GLOBALCONSTANTS DefaultPool (* Global constants *)
  PACKAGE FBs::Counter::const;
  VAR_GLOBAL CONSTANT
    ISO_DESIGNATOR_WIDTH : UINT := 80;
    ISO_DESIGNATOR_HEIGHT : UINT := 80;
    ISO_MASK_SIZE : UINT := 480;
    ISO_VERSION_LABEL : STRING;
    MASK_WIDTH : UINT := 480;
    MASK_HEIGHT : UINT := 480;
    WorkingSet : UINT := 0;
    DataMask_Home : UINT := 1000;
    Container_Gesamtzaehler : UINT := 3000;
    Container_Tageszaehler : UINT := 3001;
    SoftKeyMask_Home : UINT := 4000;
    SoftKey_PlusPlus : UINT := 5000;
    SoftKey_Reset_Gesamtzaehler : UINT := 5001;
    SoftKey_Reset_Tageszaehler : UINT := 5002;
    SoftKey_MinusMinus : UINT := 5003;
    Button_PlusPlus : UINT := 6000;
    Button_Reset_Gesamtzaehler : UINT := 6001;
    Button_Reset_Tageszaehler : UINT := 6002;
    Button_MinusMinus : UINT := 6003;
    Button_NextVT : UINT := 6004;
    InputNumber_Gesamtziel : UINT := 9000;
    InputNumber_Tagesziel : UINT := 9001;
    OutputString_NextVT : UINT := 11000;
    OutputString_Fasszaehler : UINT := 11001;
    OutputString_Reset_Gesamtzaehler : UINT := 11002;
    OutputString_Gesamtzaehler : UINT := 11003;
    OutputString_Tageszaehler : UINT := 11004;
    OutputString_Reset_Tageszaehler : UINT := 11005;
    OutputString_SoftKey_Reset_Gesamtzaehler : UINT := 11009;
    OutputString_SoftKey_Reset_Tageszaehler : UINT := 11010;
    OutputString_Ziel : UINT := 11011;
    OutputString_ZielErreicht : UINT := 11012;
    OutputNumber_Tageszaehler : UINT := 12000;
    OutputNumber_Gesamtzaehler : UINT := 12003;
    Rectangle_Box : UINT := 14000;
    Meter_Gesamtzaehler : UINT := 17000;
    Meter_Tageszaehler : UINT := 17001;
    LinearBargraph_Gesamtzaehler : UINT := 18000;
    LinearBargraph_Tageszaehler : UINT := 18001;
    Icon_Button_MinusMinus : UINT := 20000;
    Icon_Button_PlusPlus : UINT := 20001;
    Icon_SoftKey_MinusMinus : UINT := 20002;
    IconSoftKey_PlusPlus : UINT := 20003;
    NumberVariable_Tageszaehler : UINT := 21000;
    NumberVariable_Gesamtzaehler : UINT := 21001;
    NumberVariable_Gesamtziel : UINT := 21002;
    NumberVariable_Tagesziel : UINT := 21003;
    FontAttributes_Default : UINT := 23001;
    FontAttributes_Button : UINT := 23002;
    LineAttributes_Border : UINT := 24000;
    FillAttributes_DarkerBG : UINT := 25000;
    ObjectPointer_Null2 : UINT := 27000;
    ObjectPointer_Tagesziel : UINT := 27001;
    ObjectPointer_Gesamtziel : UINT := 27003;
    AuxFunction2_PlusPlus : UINT := 31000;
    AuxFunction2_MinusMinus : UINT := 31001;
  END_VAR
END_GLOBALCONSTANTS
